{attribute 'no_explicit_call' := 'do not call this POU directly, call execute'} 
FUNCTION_BLOCK _TemplateFB_1
VAR
END_VAR

// NO CODE HERE, USE execute

METHOD execute
END_METHOD

END_FUNCTION_BLOCK

(* stored: Version 1.1.0.1
   POU _TemplateFB_1: Id {2323263b-6f73-4322-9918-d8512b5e00f4}, SpecialFunc None
   Method execute: Id {cbc726b1-62f0-4983-a529-a06c892c6489} *)
